{attribute 'linkalways'} 
{attribute 'no_explicit_call' := 'This FB is a CLASS and must be accessed using methods or properties'}
{attribute 'enable_dynamic_creation'}
FUNCTION_BLOCK FINAL MUL_LWORD EXTENDS Node
VAR
	in1 : _LWORD(0);
	in2 : _LWORD(0);
	out : _LWORD(0);
END_VAR

METHOD PUBLIC Clone : I_Node
VAR
	pNode : POINTER TO MUL_LWORD;
END_VAR
pNode := __NEW(MUL_LWORD);
Clone := pNode^;
END_METHOD

METHOD FB_init : BOOL
VAR_INPUT
	bInitRetains : BOOL; // if TRUE, the retain variables are initialized (warm start / cold start)
	bInCopyCode : BOOL;  // if TRUE, the instance afterwards gets moved into the copy code (online change)
END_VAR
AddInput('in1',THIS^.in1);
AddInput('in2',THIS^.in2);
AddOutput('out', THIS^.out);
END_METHOD

METHOD PROTECTED OnExecute
VAR
END_VAR
out.Value := in1.Value * in2.Value;
END_METHOD

END_FUNCTION_BLOCK

(* stored: Version 1.1.0.1, ProductVersion 3.1.4024.15
   POU MUL_LWORD: Id {5d7c9b3b-ddd5-4dfd-a724-467d5ee5bdda}, SpecialFunc None
   Folder Constructor: Id {193bafd4-55b7-4b27-8475-9e3d03566d26}
   Method Clone: Id {177d3dc6-095a-4074-95bd-60744e0a4399}
   Method FB_init: Id {ac7eb169-d272-439d-9a30-7d918f2345fe}
   Method OnExecute: Id {d11cff8b-c077-4cc2-b844-75643644acde} *)
